(* PLC project desalination, Generated TextualNotationConverter 1.0 *)
(* stored: creationDateTime 2025-07-30T12:00:00, modificationDateTime 2025-01-30T12:00:00 *)

FUNCTION_BLOCK ANALOG_IN
  VAR_INPUT
    Name : STRING;
    Description : STRING;
    Raw_Signal : REAL;
    PV_High : REAL;
    PV_Low : REAL;
    Scaling_Slope : REAL;
    Scaling_Offset : REAL;
    Alarm_Enable : BOOL;
  END_VAR
  VAR_OUTPUT
    PV : REAL;
    High_Alarm : BOOL;
    Low_Alarm : BOOL;
    General_Fault : BOOL;
  END_VAR

            
          
END_FUNCTION_BLOCK

FUNCTION_BLOCK PID_BASIC
  VAR_INPUT
    Name : STRING;
    Description : STRING;
    AUTO : BOOL;
    PV : REAL;
    SP : REAL;
    MV_MIN : REAL;
    MV_MAX : REAL;
    X0 : REAL;
    KP : REAL;
    TR : REAL;
    TD : REAL;
    PV_High : REAL;
    PV_Low : REAL;
    Deviation_Limit : REAL;
    Inhibit : BOOL;
  END_VAR
  VAR_OUTPUT
    PV_High_Alarm : BOOL;
    PV_Low_Alarm : BOOL;
    Deviation_Alarm : BOOL;
    XOUT : REAL;
  END_VAR

            
          
END_FUNCTION_BLOCK

FUNCTION_BLOCK VALVE_ELECTRIC
  VAR_INPUT
    Name : STRING;
    Description : STRING;
    Control_Signal : REAL;
    Manual_Mode : BOOL;
    Manual_Position : REAL;
    Open_Limit : REAL;
    Close_Limit : REAL;
    Timeout : STRING;
    Inhibit : BOOL;
  END_VAR
  VAR_OUTPUT
    Valve_Position : REAL;
    Feedback_Pos : REAL;
    Valve_Moving : BOOL;
    Position_Error : BOOL;
    Alarm : BOOL;
  END_VAR

            
          
END_FUNCTION_BLOCK

FUNCTION_BLOCK VALVE_ON_OFF
  VAR_INPUT
    Name : STRING;
    Description : STRING;
    Open_Cmd : BOOL;
    Close_Cmd : BOOL;
    Timeout : STRING;
    Inhibit : BOOL;
  END_VAR
  VAR_OUTPUT
    FB_Opened : BOOL;
    FB_Closed : BOOL;
    Valve_Open_Out : BOOL;
    Valve_Close_Out : BOOL;
    Alarm_Position_Error : BOOL;
    Alarm_General : BOOL;
  END_VAR

            
          
END_FUNCTION_BLOCK

PROGRAM Section2
  VAR
    FT101_Flow_PV : REAL;
    FT102_Flow_PV : REAL;
    AT101_Analyzer_PV : REAL;
    AT103_Analyzer_PV : REAL;
    LT104_Level_PV : REAL;
    LT105_Level_PV : REAL;
    FC101_MV_Out : REAL;
    FC102_MV_Out : REAL;
    FV101_Valve_Position : REAL;
    FV102_Valve_Position : REAL;
    SP101_PctCmd : REAL;
    SP102_PctCmd : REAL;
    FlowDevAlarm101 : BOOL;
    FlowDevAlarm102 : BOOL;
  END_VAR
  VAR
    AT-101 : ANALOG_IN;
    AT-103 : ANALOG_IN;
    FC-101 : PID_BASIC;
    FC-102 : PID_BASIC;
    FT-101 : ANALOG_IN;
    FT-102 : ANALOG_IN;
    FV-101 : VALVE_ELECTRIC;
    FV-102 : VALVE_ELECTRIC;
    LT-104 : ANALOG_IN;
    LT-105 : ANALOG_IN;
    XV-102 : VALVE_ON_OFF;
    SP101_DevDelay_TON : TON;
    SP102_DevDelay_TON : TON;
  END_VAR
  VAR  (* added by the conversion: wires and edge detectors of the diagram *)
    _MULT9_OUT : REAL;
    _MULT20_OUT : REAL;
    _OR2_OUT : BOOL;
    _NOT1_OUT : BOOL;
  END_VAR

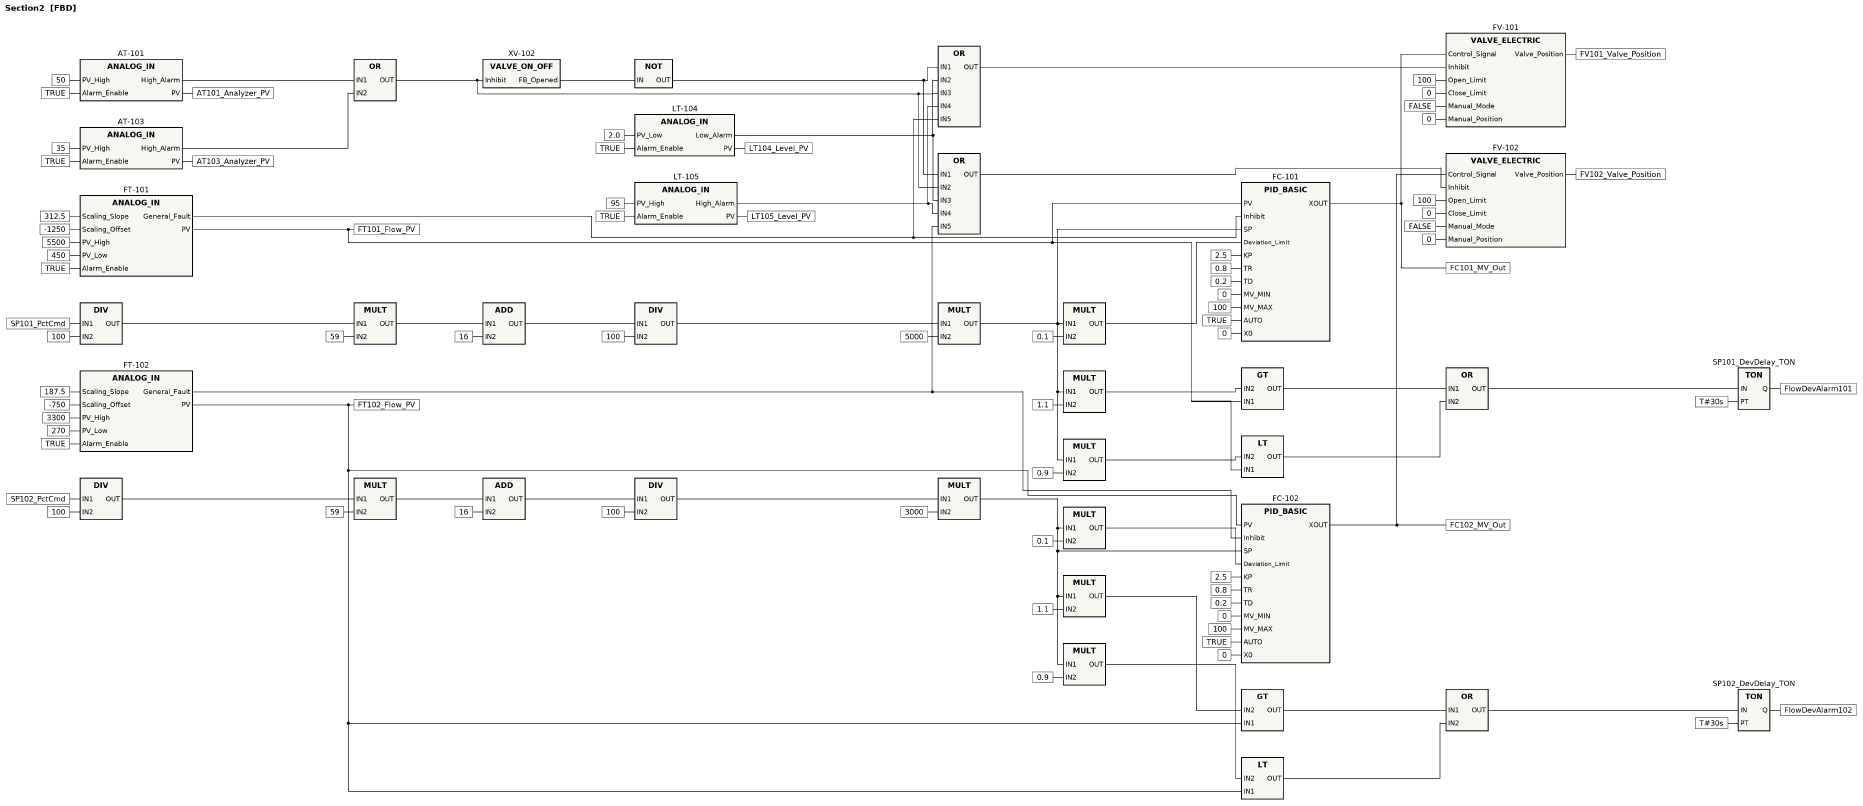
(* FBD diagram, written out as Structured Text *)
AT-101(PV_High := 50, Alarm_Enable := TRUE);
AT101_Analyzer_PV := AT-101.PV;
AT-103(PV_High := 35, Alarm_Enable := TRUE);
AT103_Analyzer_PV := AT-103.PV;
FT-101(Scaling_Slope := 312.5, Scaling_Offset := -1250, PV_High := 5500, PV_Low := 450, Alarm_Enable := TRUE);
_MULT9_OUT := MULT((MULT(SP101_PctCmd / 100, 59) + 16) / 100, 5000);
FC-101(PV := FT-101.PV, Inhibit := FT-101.General_Fault, SP := _MULT9_OUT, Deviation_Limit := MULT(_MULT9_OUT, 0.1), KP := 2.5, TR := 0.8, TD := 0.2, MV_MIN := 0, MV_MAX := 100, AUTO := TRUE, X0 := 0);
FC101_MV_Out := FC-101.XOUT;
FT-102(Scaling_Slope := 187.5, Scaling_Offset := -750, PV_High := 3300, PV_Low := 270, Alarm_Enable := TRUE);
_MULT20_OUT := MULT((MULT(SP102_PctCmd / 100, 59) + 16) / 100, 3000);
FC-102(PV := FT-102.PV, Inhibit := FT-102.General_Fault, SP := _MULT20_OUT, Deviation_Limit := MULT(_MULT20_OUT, 0.1), KP := 2.5, TR := 0.8, TD := 0.2, MV_MIN := 0, MV_MAX := 100, AUTO := TRUE, X0 := 0);
FC102_MV_Out := FC-102.XOUT;
FT101_Flow_PV := FT-101.PV;
FT102_Flow_PV := FT-102.PV;
_OR2_OUT := AT-101.High_Alarm OR AT-103.High_Alarm;
XV-102(Inhibit := _OR2_OUT);
_NOT1_OUT := NOT XV-102.FB_Opened;
LT-104(PV_Low := 2.0, Alarm_Enable := TRUE);
LT-105(PV_High := 95, Alarm_Enable := TRUE);
FV-101(Control_Signal := FC-101.XOUT, Inhibit := _NOT1_OUT OR _OR2_OUT OR LT-104.Low_Alarm OR LT-105.High_Alarm OR FT-101.General_Fault, Open_Limit := 100, Close_Limit := 0, Manual_Mode := FALSE, Manual_Position := 0);
FV101_Valve_Position := FV-101.Valve_Position;
FV-102(Control_Signal := FC-102.XOUT, Inhibit := _NOT1_OUT OR _OR2_OUT OR LT-104.Low_Alarm OR LT-105.High_Alarm OR FT-102.General_Fault, Open_Limit := 100, Close_Limit := 0, Manual_Mode := FALSE, Manual_Position := 0);
FV102_Valve_Position := FV-102.Valve_Position;
SP101_DevDelay_TON(IN := MULT(_MULT9_OUT, 1.1) > FT-101.PV OR MULT(_MULT9_OUT, 0.9) < FT-101.PV, PT := T#30s);
FlowDevAlarm101 := SP101_DevDelay_TON.Q;
SP102_DevDelay_TON(IN := MULT(_MULT20_OUT, 1.1) > FT-102.PV OR MULT(_MULT20_OUT, 0.9) < FT-102.PV, PT := T#30s);
FlowDevAlarm102 := SP102_DevDelay_TON.Q;
LT104_Level_PV := LT-104.PV;
LT105_Level_PV := LT-105.PV;
END_PROGRAM

FUNCTION_BLOCK BOOL_IN
  VAR_INPUT
    Name : STRING;
    Description : STRING;
    Bool_In : BOOL;
    Alarm_OnTrue : BOOL;
    Alarm_OnFalse : BOOL;
    Latch_Enable : BOOL;
    Reset_Latch : BOOL;
  END_VAR
  VAR_OUTPUT
    Bool_Out : BOOL;
    Alarm_Active : BOOL;
    Latched_Status : BOOL;
  END_VAR

            
          
END_FUNCTION_BLOCK

FUNCTION_BLOCK DIGITAL_IN
  VAR_INPUT
    Name : STRING;
    Description : STRING;
    DI_Raw : BOOL;
    DebounceTime : STRING;
    EnableAlarm : BOOL;
  END_VAR
  VAR_OUTPUT
    DI_Out : BOOL;
    Fault_State : BOOL;
  END_VAR

            
          
END_FUNCTION_BLOCK

FUNCTION_BLOCK DUTY_STANDBY
  VAR_INPUT
    Name : STRING;
    Description : STRING;
    Enable : BOOL;
    StartRequest : BOOL;
    AlternateEnable : BOOL;
    ForcePumpA : BOOL;
    ForcePumpB : BOOL;
    DutyElapsed : BOOL;
    MinRunElapsed : BOOL;
    SwitchoverDelayElapsed : BOOL;
    StartTimeoutElapsed : BOOL;
    PumpA_RunFB : BOOL;
    PumpB_RunFB : BOOL;
    PumpA_Fault : BOOL;
    PumpB_Fault : BOOL;
    Reset : BOOL;
    Inhibit : BOOL;
  END_VAR
  VAR_OUTPUT
    CmdPumpA : BOOL;
    CmdPumpB : BOOL;
    ActiveIsA : BOOL;
    SwitchedDueToDuty : BOOL;
    SwitchedDueToFailure : BOOL;
    Alarm_FailedStart_A : BOOL;
    Alarm_FailedStart_B : BOOL;
    Alarm_NoAvailablePump : BOOL;
  END_VAR

            
          
END_FUNCTION_BLOCK

FUNCTION_BLOCK MOTOR_2SPD
  VAR_INPUT
    Name : STRING;
    Description : STRING;
    Start_Cmd : BOOL;
    Stop_Cmd : BOOL;
    Speed_High_Cmd : BOOL;
    Speed_Low_Cmd : BOOL;
    Inhibit : BOOL;
  END_VAR
  VAR_OUTPUT
    Motor_Start_Out : BOOL;
    FB_Running : BOOL;
    FB_Trip : BOOL;
    FB_HighSpeed : BOOL;
    FB_LowSpeed : BOOL;
    Alarm_Speed_Error : BOOL;
  END_VAR

            
          
END_FUNCTION_BLOCK

FUNCTION_BLOCK MOTOR_ON_OFF
  VAR_INPUT
    Name : STRING;
    Description : STRING;
    Start_Cmd : BOOL;
    Stop_Cmd : BOOL;
    Start_Delay : STRING;
    MinRunTime : STRING;
    Inhibit : BOOL;
  END_VAR
  VAR_OUTPUT
    Motor_Start_Out : BOOL;
    FB_Running : BOOL;
    FB_Trip : BOOL;
    Alarm_Start_Fail : BOOL;
    Alarm_Stop_Fail : BOOL;
  END_VAR

            
          
END_FUNCTION_BLOCK

FUNCTION_BLOCK MOTOR_VSD
  VAR_INPUT
    Name : STRING;
    Description : STRING;
    Start_Cmd : BOOL;
    Stop_Cmd : BOOL;
    Speed_SP : REAL;
    Accel_Ramp : STRING;
    Decel_Ramp : STRING;
    Inhibit : BOOL;
  END_VAR
  VAR_OUTPUT
    Speed_Out : REAL;
    FB_Running : BOOL;
    FB_Fault : BOOL;
    FB_Ready : BOOL;
    FB_ActualSpeed : REAL;
    Alarm_Speed_Deviation : BOOL;
    Alarm_Comm_Fail : BOOL;
  END_VAR

            
          
END_FUNCTION_BLOCK

FUNCTION_BLOCK RATIO_CONTROL
  VAR_INPUT
    Name : STRING;
    Description : STRING;
    Auto : BOOL;
    PrimaryPV : REAL;
    SecondaryPV : REAL;
    RatioSP : REAL;
    Bias : REAL;
    TrimKp : REAL;
    TrimTi : STRING;
    MV_MIN : REAL;
    MV_MAX : REAL;
    ManOut : REAL;
    Inhibit : BOOL;
  END_VAR
  VAR_OUTPUT
    SlaveSP : REAL;
    ActiveRatio : REAL;
    RatioErr : REAL;
  END_VAR

            
          
END_FUNCTION_BLOCK

FUNCTION_BLOCK SPLIT_RANGE
  VAR_INPUT
    Name : STRING;
    Description : STRING;
    IN : REAL;
    Split_Point : REAL;
    Output1_Start : REAL;
    Output1_End : REAL;
    Output2_Start : REAL;
    Output2_End : REAL;
  END_VAR
  VAR_OUTPUT
    OUT1 : REAL;
    OUT2 : REAL;
  END_VAR

            
          
END_FUNCTION_BLOCK

FUNCTION_BLOCK VOTING_ANALOG
  VAR_INPUT
    Name : STRING;
    Description : STRING;
    Input1 : REAL;
    Input2 : REAL;
    Input3 : REAL;
    Deviation_Limit : REAL;
    Voting_Scheme : STRING;
    EnableAlarm : BOOL;
    Inhibit : BOOL;
  END_VAR
  VAR_OUTPUT
    Voted_Output : REAL;
    Sensor1_Fault : BOOL;
    Sensor2_Fault : BOOL;
    Sensor3_Fault : BOOL;
    Alarm_Voting_Error : BOOL;
    Healthy_Sensors_Count : INT;
  END_VAR

            
          
END_FUNCTION_BLOCK

PROGRAM Section3
  VAR
    FT102_SP_FromRatio : REAL;
    FV105_Feedback_Position : REAL;
  END_VAR
  VAR
    FFIC-103 : RATIO_CONTROL;
    FIC-104 : PID_BASIC;
    FV-105 : VALVE_ELECTRIC;
    FT-101 : ANALOG_IN;
    FT-102 : ANALOG_IN;
    PT-103 : ANALOG_IN;
    PT-104 : ANALOG_IN;
    PIT-105 : ANALOG_IN;
    PIT-106 : ANALOG_IN;
    PT-108 : ANALOG_IN;
    SW-SCREEN-1 : BOOL_IN;
    SW-SCREEN-2 : BOOL_IN;
    SW-SCREEN-3 : BOOL_IN;
    SW-SCREEN-4 : BOOL_IN;
    SW-SCREEN-5 : BOOL_IN;
    SW-SCREEN-6 : BOOL_IN;
    RES-SCREEN-1 : BOOL_IN;
    RES-SCREEN-2 : BOOL_IN;
    RES-SCREEN-3 : BOOL_IN;
    RES-SCREEN-4 : BOOL_IN;
  END_VAR
  VAR  (* added by the conversion: wires and edge detectors of the diagram *)
    _RS114_OUT : BOOL;
    _OR116_OUT : BOOL;
    _OR117_OUT : BOOL;
  END_VAR

(* FBD diagram, written out as Structured Text *)
FT-101(Scaling_Slope := 31.25, Scaling_Offset := -125.0, PV_Low := 50.0, Alarm_Enable := TRUE);
FT-102(Scaling_Slope := 31.25, Scaling_Offset := -125.0);
_RS114_OUT := RS(FT-101.PV < 50.0, FT-101.PV > 50.0);
PT-103(Low_Alarm := FT-101.PV, PV_Low := 6.0, Alarm_Enable := TRUE);
PIT-105(PV_Low := 4.0, PV_High := 8.0, Alarm_Enable := TRUE);
PIT-106(PV_Low := 4.0, PV_High := 8.0, Alarm_Enable := TRUE);
_OR116_OUT := PIT-105.Low_Alarm OR PIT-105.High_Alarm OR PIT-106.Low_Alarm OR PIT-106.High_Alarm;
PT-108(PV_Low := 5.0, PV_High := 9.0, Alarm_Enable := TRUE);
_OR117_OUT := PT-108.Low_Alarm OR PT-108.High_Alarm;
FIC-104(SP := FFIC-103.SlaveSP, PV := FT-102.PV, AUTO := NOT _RS114_OUT);
FV-105(Control_Signal := FIC-104.XOUT, Inhibit := _OR116_OUT OR _OR117_OUT, Timeout := T#2s);
SW-SCREEN-1();
SW-SCREEN-2();
SW-SCREEN-3();
SW-SCREEN-4();
SW-SCREEN-5();
SW-SCREEN-6();
RES-SCREEN-1();
RES-SCREEN-2();
RES-SCREEN-3();
RES-SCREEN-4();
PT-104(Low_Alarm := FT-101.PV, PV_Low := 6.0, Alarm_Enable := TRUE);
FFIC-103(PrimaryPV := FT-101.PV, SecondaryPV := FT-102.PV, Inhibit := _RS114_OUT OR PT-103.Low_Alarm OR _OR116_OUT OR _OR117_OUT OR FV-105.Position_Error OR SW-SCREEN-1.Bool_Out AND (SW-SCREEN-2.Bool_Out OR SW-SCREEN-3.Bool_Out OR SW-SCREEN-4.Bool_Out OR SW-SCREEN-5.Bool_Out OR SW-SCREEN-6.Bool_Out OR RES-SCREEN-1.Bool_Out OR RES-SCREEN-2.Bool_Out OR RES-SCREEN-3.Bool_Out OR RES-SCREEN-4.Bool_Out) OR SW-SCREEN-2.Bool_Out AND (SW-SCREEN-1.Bool_Out OR SW-SCREEN-3.Bool_Out OR SW-SCREEN-4.Bool_Out OR SW-SCREEN-5.Bool_Out OR SW-SCREEN-6.Bool_Out OR RES-SCREEN-1.Bool_Out OR RES-SCREEN-2.Bool_Out OR RES-SCREEN-3.Bool_Out OR RES-SCREEN-4.Bool_Out) OR SW-SCREEN-3.Bool_Out AND (SW-SCREEN-1.Bool_Out OR SW-SCREEN-2.Bool_Out OR SW-SCREEN-4.Bool_Out OR SW-SCREEN-5.Bool_Out OR SW-SCREEN-6.Bool_Out OR RES-SCREEN-1.Bool_Out OR RES-SCREEN-2.Bool_Out OR RES-SCREEN-3.Bool_Out OR RES-SCREEN-4.Bool_Out) OR SW-SCREEN-4.Bool_Out AND (SW-SCREEN-1.Bool_Out OR SW-SCREEN-2.Bool_Out OR SW-SCREEN-3.Bool_Out OR SW-SCREEN-5.Bool_Out OR SW-SCREEN-6.Bool_Out OR RES-SCREEN-1.Bool_Out OR RES-SCREEN-2.Bool_Out OR RES-SCREEN-3.Bool_Out OR RES-SCREEN-4.Bool_Out) OR SW-SCREEN-5.Bool_Out AND (SW-SCREEN-1.Bool_Out OR SW-SCREEN-2.Bool_Out OR SW-SCREEN-3.Bool_Out OR SW-SCREEN-4.Bool_Out OR SW-SCREEN-6.Bool_Out OR RES-SCREEN-1.Bool_Out OR RES-SCREEN-2.Bool_Out OR RES-SCREEN-3.Bool_Out OR RES-SCREEN-4.Bool_Out) OR SW-SCREEN-6.Bool_Out AND (SW-SCREEN-1.Bool_Out OR SW-SCREEN-2.Bool_Out OR SW-SCREEN-3.Bool_Out OR SW-SCREEN-4.Bool_Out OR SW-SCREEN-5.Bool_Out OR RES-SCREEN-1.Bool_Out OR RES-SCREEN-2.Bool_Out OR RES-SCREEN-3.Bool_Out OR RES-SCREEN-4.Bool_Out) OR RES-SCREEN-1.Bool_Out AND (SW-SCREEN-1.Bool_Out OR SW-SCREEN-2.Bool_Out OR SW-SCREEN-3.Bool_Out OR SW-SCREEN-4.Bool_Out OR SW-SCREEN-5.Bool_Out OR SW-SCREEN-6.Bool_Out OR RES-SCREEN-2.Bool_Out OR RES-SCREEN-3.Bool_Out OR RES-SCREEN-4.Bool_Out) OR RES-SCREEN-2.Bool_Out AND (SW-SCREEN-1.Bool_Out OR SW-SCREEN-2.Bool_Out OR SW-SCREEN-3.Bool_Out OR SW-SCREEN-4.Bool_Out OR SW-SCREEN-5.Bool_Out OR SW-SCREEN-6.Bool_Out OR RES-SCREEN-1.Bool_Out OR RES-SCREEN-3.Bool_Out OR RES-SCREEN-4.Bool_Out) OR RES-SCREEN-3.Bool_Out AND (SW-SCREEN-1.Bool_Out OR SW-SCREEN-2.Bool_Out OR SW-SCREEN-3.Bool_Out OR SW-SCREEN-4.Bool_Out OR SW-SCREEN-5.Bool_Out OR SW-SCREEN-6.Bool_Out OR RES-SCREEN-1.Bool_Out OR RES-SCREEN-2.Bool_Out OR RES-SCREEN-4.Bool_Out) OR RES-SCREEN-4.Bool_Out AND (SW-SCREEN-1.Bool_Out OR SW-SCREEN-2.Bool_Out OR SW-SCREEN-3.Bool_Out OR SW-SCREEN-4.Bool_Out OR SW-SCREEN-5.Bool_Out OR SW-SCREEN-6.Bool_Out OR RES-SCREEN-1.Bool_Out OR RES-SCREEN-2.Bool_Out OR RES-SCREEN-3.Bool_Out) OR FIC-104.Deviation_Alarm OR PT-104.Low_Alarm, RatioSP := 2.0, MV_MIN := 0.0, MV_MAX := 500.0);
FT102_SP_FromRatio := FFIC-103.SlaveSP;
FV105_Feedback_Position := FV-105.Feedback_Pos;
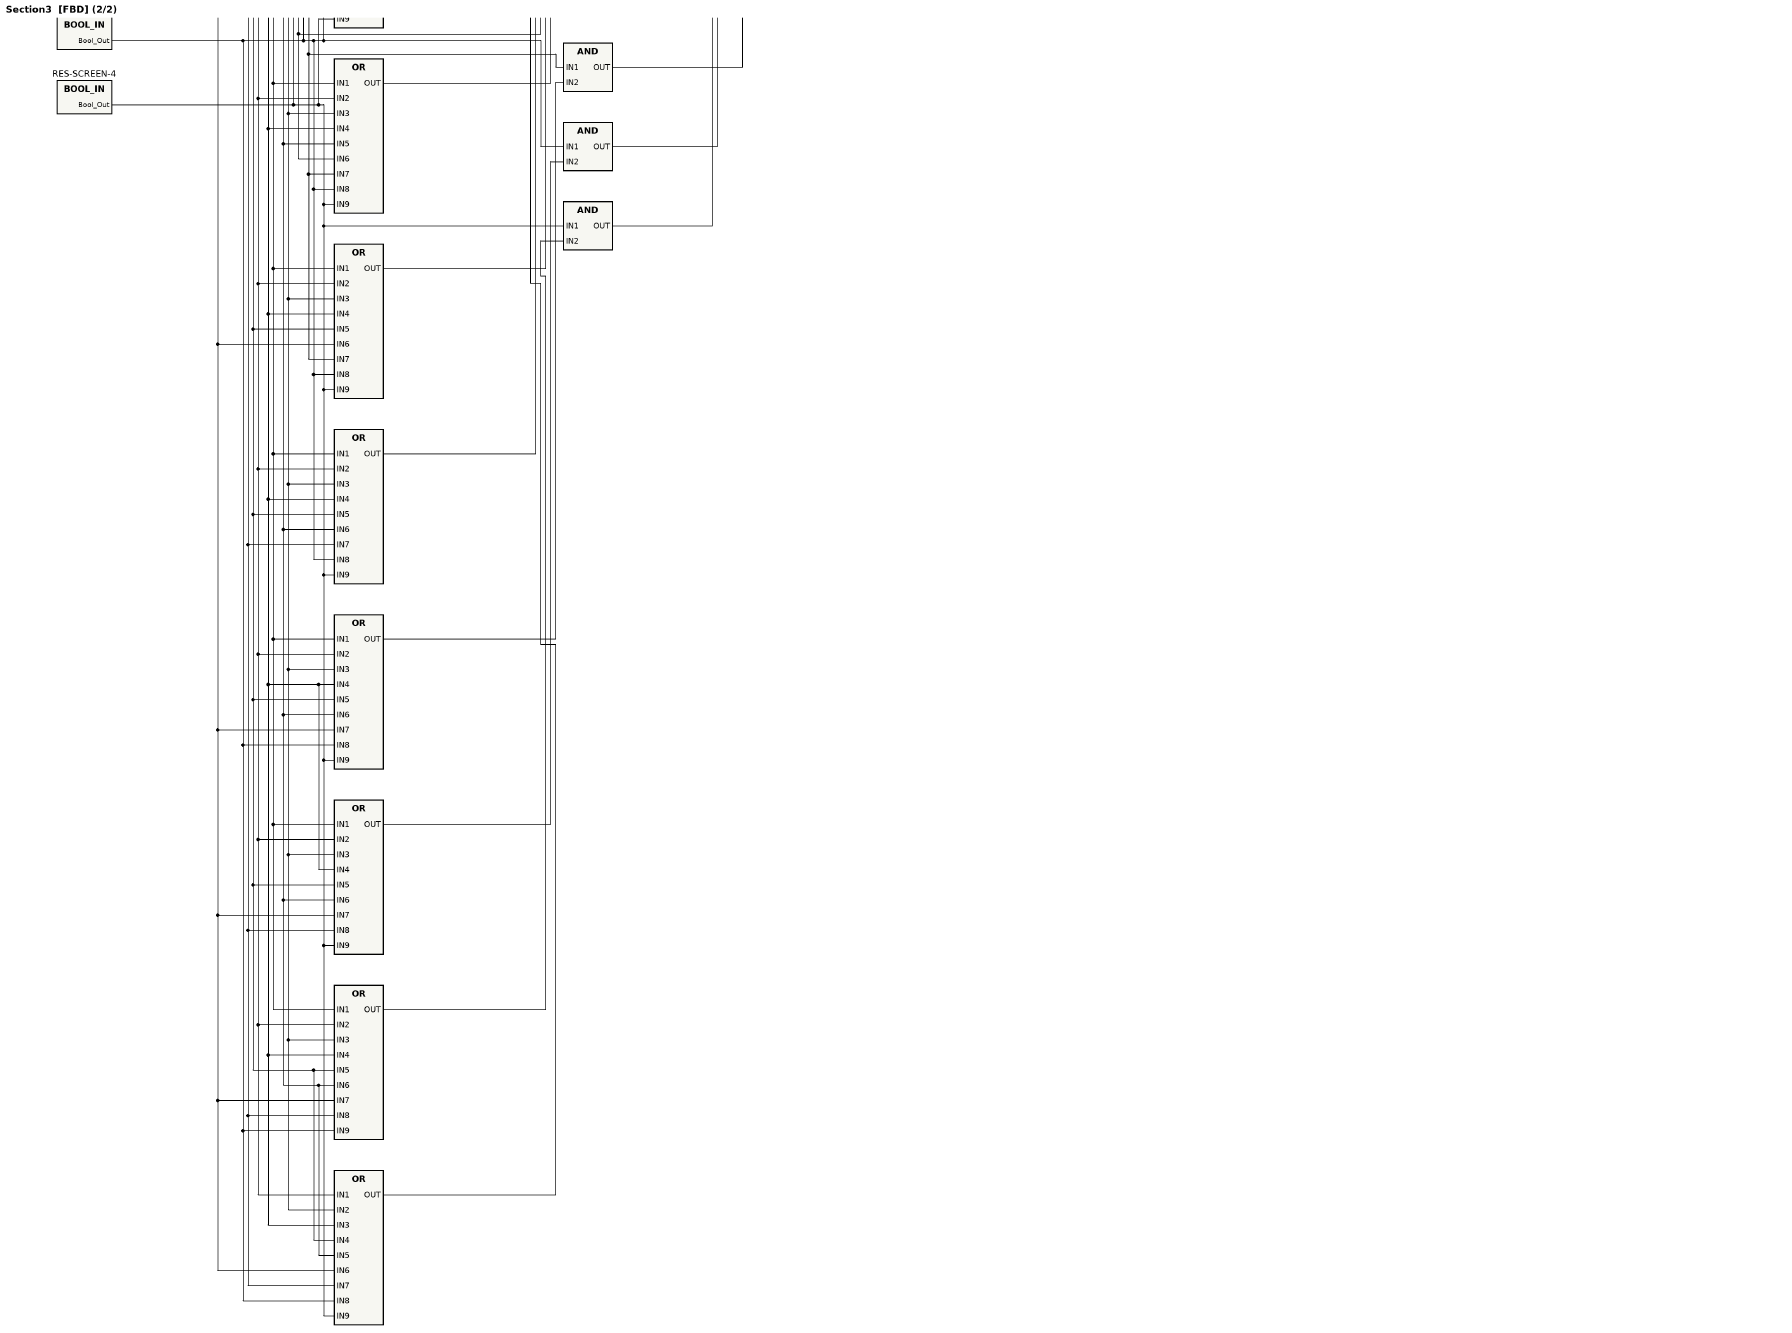
END_PROGRAM

PROGRAM Section4
  VAR
    FT_101_Flow_PV_m3ph : REAL;
    LT_101_SumpLevel_m : REAL;
    FIC_101_MV_Percent : REAL;
    FIC_101_SP_m3ph : REAL;
    Flow_Deviation_Alarm : BOOL;
  END_VAR
  VAR
    FT-101 : ANALOG_IN;
    LT-101 : ANALOG_IN;
    FIC-101 : PID_BASIC;
    VFD-101A : MOTOR_VSD;
    VFD-101B : MOTOR_VSD;
    VFD-101C : MOTOR_VSD;
    VFD-101D : MOTOR_VSD;
    SPUMP-201A : MOTOR_ON_OFF;
    SPUMP-201B : MOTOR_ON_OFF;
    M103A : DIGITAL_IN;
    M103B : DIGITAL_IN;
    M103C : DIGITAL_IN;
    M103D : DIGITAL_IN;
    FlowDeviationHold : TON;
  END_VAR
  VAR  (* added by the conversion: wires and edge detectors of the diagram *)
    _OR188_OUT : BOOL;
    _OR189_OUT : BOOL;
    _OR190_OUT : BOOL;
    _OR191_OUT : BOOL;
    _OR192_OUT : BOOL;
  END_VAR

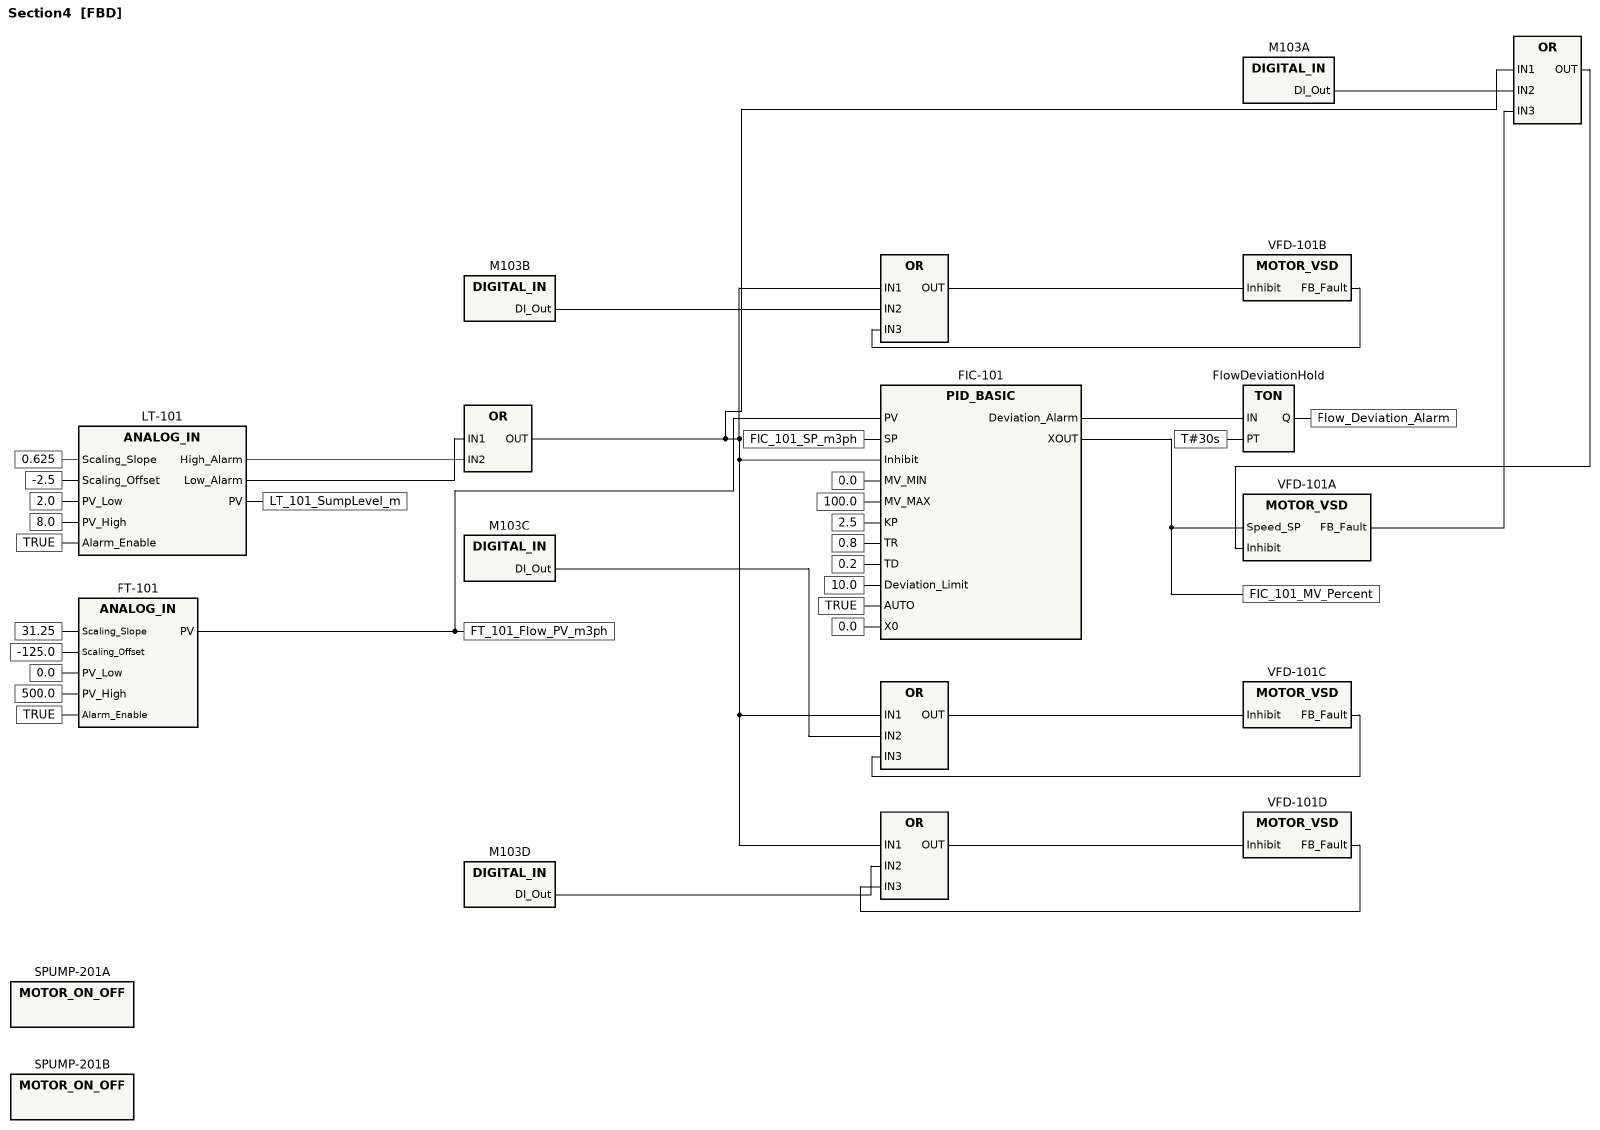
(* FBD diagram, written out as Structured Text *)
FT-101(Scaling_Slope := 31.25, Scaling_Offset := -125.0, PV_Low := 0.0, PV_High := 500.0, Alarm_Enable := TRUE);
LT-101(Scaling_Slope := 0.625, Scaling_Offset := -2.5, PV_Low := 2.0, PV_High := 8.0, Alarm_Enable := TRUE);
_OR188_OUT := LT-101.Low_Alarm OR LT-101.High_Alarm;
FIC-101(PV := FT-101.PV, SP := FIC_101_SP_m3ph, Inhibit := _OR188_OUT, MV_MIN := 0.0, MV_MAX := 100.0, KP := 2.5, TR := 0.8, TD := 0.2, Deviation_Limit := 10.0, AUTO := TRUE, X0 := 0.0);
FIC_101_MV_Percent := FIC-101.XOUT;
FT_101_Flow_PV_m3ph := FT-101.PV;
FlowDeviationHold(IN := FIC-101.Deviation_Alarm, PT := T#30s);
Flow_Deviation_Alarm := FlowDeviationHold.Q;
LT_101_SumpLevel_m := LT-101.PV;
M103A();
VFD-101A(Speed_SP := FIC-101.XOUT, Inhibit := _OR189_OUT);
_OR189_OUT := _OR188_OUT OR M103A.DI_Out OR VFD-101A.FB_Fault;
M103B();
VFD-101B(Inhibit := _OR190_OUT);
_OR190_OUT := _OR188_OUT OR M103B.DI_Out OR VFD-101B.FB_Fault;
M103C();
VFD-101C(Inhibit := _OR191_OUT);
_OR191_OUT := _OR188_OUT OR M103C.DI_Out OR VFD-101C.FB_Fault;
M103D();
VFD-101D(Inhibit := _OR192_OUT);
_OR192_OUT := _OR188_OUT OR M103D.DI_Out OR VFD-101D.FB_Fault;
SPUMP-201A();
SPUMP-201B();
END_PROGRAM

PROGRAM Section5
  VAR
    FT_301_FlowRate_PV : REAL;
    LT_301_Level_PV : REAL;
    FIC_301_MV_FlowControl_Percent : REAL;
    XV_107_Open_FB : BOOL;
  END_VAR
  VAR
    FT-301 : ANALOG_IN;
    LT-301 : ANALOG_IN;
    FIC-301 : PID_BASIC;
    FV-301 : VALVE_ELECTRIC;
    XV-107 : VALVE_ON_OFF;
    UMP-301A : MOTOR_VSD;
    UMP-301B : MOTOR_VSD;
    ANK-301 : BOOL_IN;
    PAH-103 : DIGITAL_IN;
    TAH-101 : DIGITAL_IN;
  END_VAR
  VAR  (* added by the conversion: wires and edge detectors of the diagram *)
    _OR235_OUT : BOOL;
    _OR236_OUT : BOOL;
  END_VAR

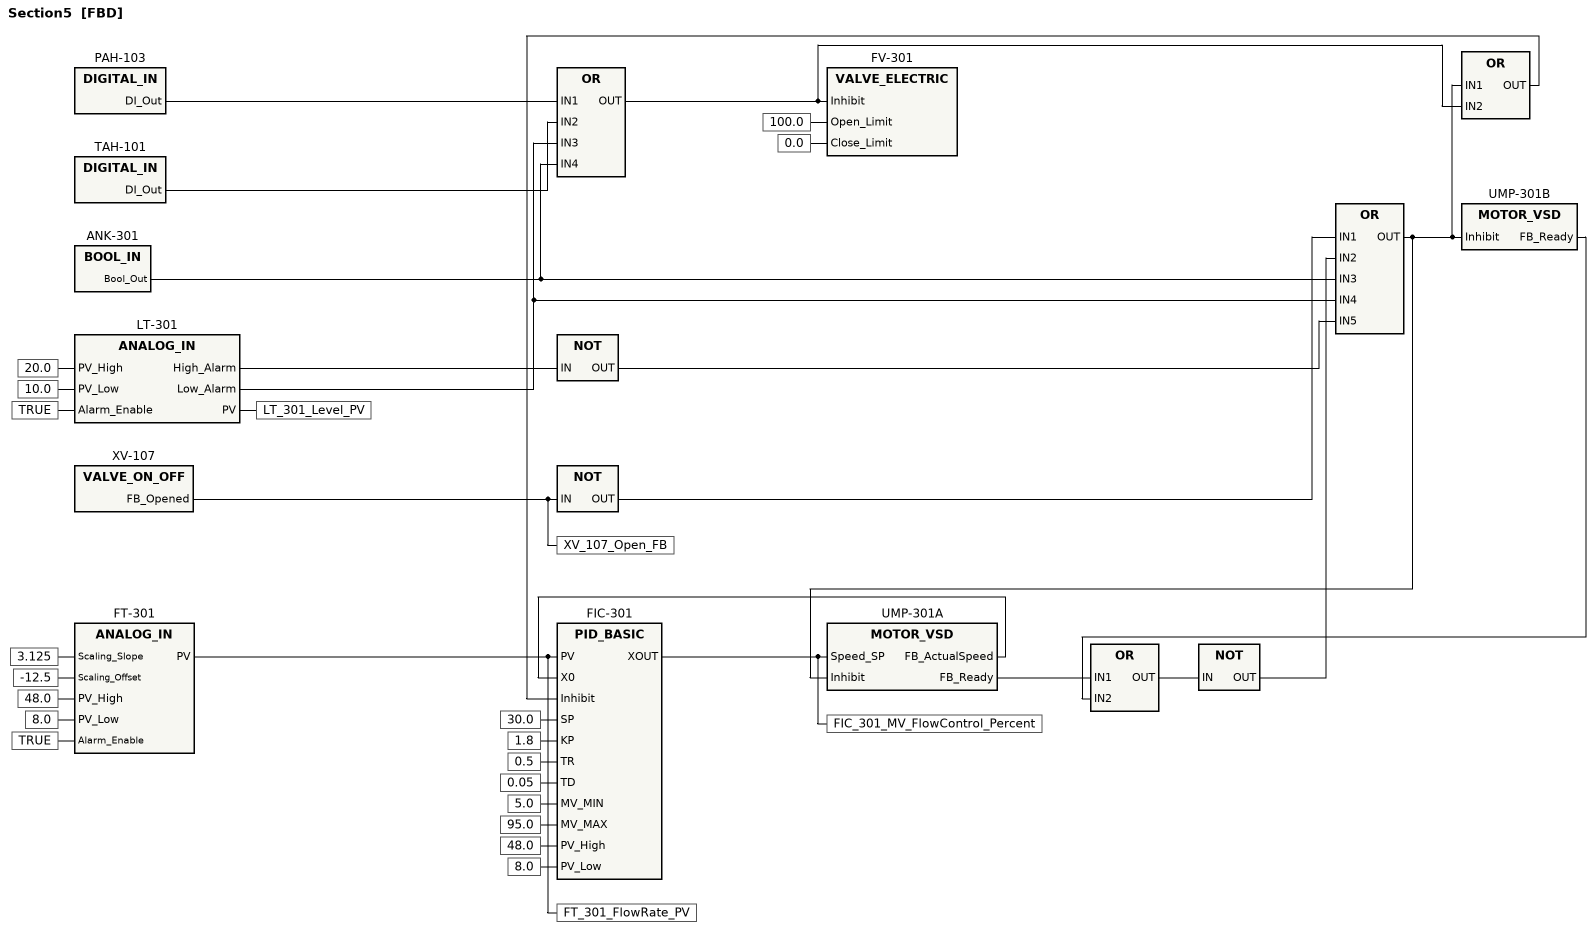
(* FBD diagram, written out as Structured Text *)
FT-301(Scaling_Slope := 3.125, Scaling_Offset := -12.5, PV_High := 48.0, PV_Low := 8.0, Alarm_Enable := TRUE);
XV-107();
UMP-301B(Inhibit := _OR235_OUT);
ANK-301();
LT-301(PV_High := 20.0, PV_Low := 10.0, Alarm_Enable := TRUE);
_OR235_OUT := NOT XV-107.FB_Opened OR NOT (UMP-301A.FB_Ready OR UMP-301B.FB_Ready) OR ANK-301.Bool_Out OR LT-301.Low_Alarm OR NOT LT-301.High_Alarm;
UMP-301A(Speed_SP := FIC-301.XOUT, Inhibit := _OR235_OUT);
PAH-103();
TAH-101();
_OR236_OUT := PAH-103.DI_Out OR TAH-101.DI_Out OR LT-301.Low_Alarm OR ANK-301.Bool_Out;
FIC-301(PV := FT-301.PV, X0 := UMP-301A.FB_ActualSpeed, Inhibit := _OR235_OUT OR _OR236_OUT, SP := 30.0, KP := 1.8, TR := 0.5, TD := 0.05, MV_MIN := 5.0, MV_MAX := 95.0, PV_High := 48.0, PV_Low := 8.0);
FIC_301_MV_FlowControl_Percent := FIC-301.XOUT;
FT_301_FlowRate_PV := FT-301.PV;
LT_301_Level_PV := LT-301.PV;
XV_107_Open_FB := XV-107.FB_Opened;
FV-301(Inhibit := _OR236_OUT, Open_Limit := 100.0, Close_Limit := 0.0);
END_PROGRAM

PROGRAM Section6
  VAR
    FIT101_BypassFlow_PV : REAL;
    FIT102_SamplingFlow_PV : REAL;
    FIC104_SamplingFlow_SP : REAL;
    FIC104_ActiveRatio : REAL;
    AT105_Permissive : BOOL;
    LV103_Permissive : BOOL;
  END_VAR
  VAR
    FIT-101 : ANALOG_IN;
    FIT-102 : ANALOG_IN;
    FIC-104 : RATIO_CONTROL;
    FIC-104_SLAVE : PID_BASIC;
    FV-102 : VALVE_ELECTRIC;
    AT-105 : BOOL_IN;
  END_VAR
  VAR  (* added by the conversion: wires and edge detectors of the diagram *)
    _OR270_OUT : BOOL;
  END_VAR

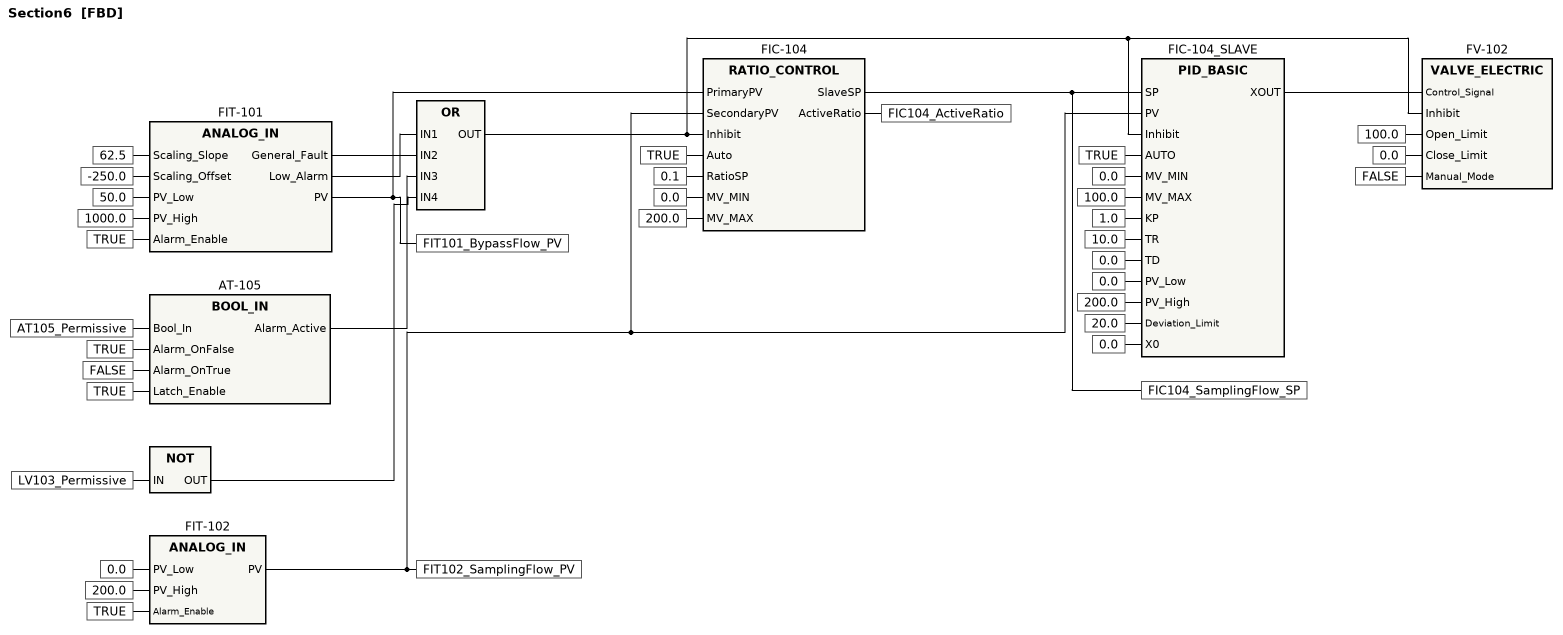
(* FBD diagram, written out as Structured Text *)
FIT-101(Scaling_Slope := 62.5, Scaling_Offset := -250.0, PV_Low := 50.0, PV_High := 1000.0, Alarm_Enable := TRUE);
FIT-102(PV_Low := 0.0, PV_High := 200.0, Alarm_Enable := TRUE);
AT-105(Bool_In := AT105_Permissive, Alarm_OnFalse := TRUE, Alarm_OnTrue := FALSE, Latch_Enable := TRUE);
_OR270_OUT := FIT-101.Low_Alarm OR FIT-101.General_Fault OR AT-105.Alarm_Active OR NOT LV103_Permissive;
FIC-104(PrimaryPV := FIT-101.PV, SecondaryPV := FIT-102.PV, Inhibit := _OR270_OUT, Auto := TRUE, RatioSP := 0.1, MV_MIN := 0.0, MV_MAX := 200.0);
FIC104_ActiveRatio := FIC-104.ActiveRatio;
FIC104_SamplingFlow_SP := FIC-104.SlaveSP;
FIT101_BypassFlow_PV := FIT-101.PV;
FIT102_SamplingFlow_PV := FIT-102.PV;
FIC-104_SLAVE(SP := FIC-104.SlaveSP, PV := FIT-102.PV, Inhibit := _OR270_OUT, AUTO := TRUE, MV_MIN := 0.0, MV_MAX := 100.0, KP := 1.0, TR := 10.0, TD := 0.0, PV_Low := 0.0, PV_High := 200.0, Deviation_Limit := 20.0, X0 := 0.0);
FV-102(Control_Signal := FIC-104_SLAVE.XOUT, Inhibit := _OR270_OUT, Open_Limit := 100.0, Close_Limit := 0.0, Manual_Mode := FALSE);
END_PROGRAM

CONFIGURATION Config0
  RESOURCE Res0 ON PLC
    TASK task0(INTERVAL := T#20ms, PRIORITY := 0);
    PROGRAM instance0 WITH task0 : Section2;
    PROGRAM instance_1 WITH task0 : Section3;
    PROGRAM instance_2 WITH task0 : Section4;
    PROGRAM instance_3 WITH task0 : Section5;
    PROGRAM instance_4 WITH task0 : Section6;
  END_RESOURCE
END_CONFIGURATION
